(* Logix 5000 project; controller MES_CORE vendor 1 type 14 code 164 rev 32.11; software revision 32.00 *)

TASK MainTask (continuous, watchdog 500 ms) : MES_CORE

MODULES
   Local : vendor 1 type 14 code 164 (ICP 0, rev 32.11)
END_MODULES

VAR_GLOBAL   (* controller tags *)
   ACTIVE_BIT : BOOL;   // FROM LINE
   ANDON : BOOL;   // FROM LINE
   E_STOP : BOOL;   // FROM LINE
   FAULT : BOOL;   // FROM LINE ACTIVE
   JAM_PE : BOOL;   // FROM LINE
   LNXX_ACTIVE_SHIFT : DINT;
   LNXX_SCHEDULE_RUNNING_ONS : BOOL[32];
   LNXX_SCHEDULED_RUN : BOOL;
   LNXX_ShiftChange : BOOL[32];
   LNXX_TO_DC01_DOWNTIME_CODE : DINT[10] := ([0] := 1036); {produced}   // DOWNTIME PRODUCE TAG
        [0]   // LN99
        [1]   // WORK CENTER MAIN LINE A
        [2]   // WORK CENTER MAIN LINE B
        [3]   // WORK CENTER MAIN LINE C
        [4]   // WORK CENTER MAIN LINE D
        [5]   // WORK CENTER MAIN LINE E
        [6]   // WORK CENTER SUB LINE C
        [7]   // WORK CENTER SUB LINE E
   LNXX_TO_DC01_MAIN_MESSAGE : DINT[20] := ([4] := 4480, [16] := 3); {produced}   // KPI PRODUCE TAGS
        [4]   // ACTUAL UNIT COUNT
        [9].0   // LINE RUNNING
        [9].1   // LINE ON BREAK
   LNXX_TO_DC1_MAIN_MESSAGE_A : DINT[10]; {produced}   // WORKCENTER A PRODUCE TAG
        [1]   // LN99NAM01
        [2]   // LN99SAM01
        [3]   // LN99NAM02
        [4]   // LN99SAM02
        [5]   // LN99NAM03
        [6]   // LN99SAM03
        [7]   // LN99NAM04
        [8]   // LN99SAM04
   RUNNING : BOOL;   // FROM LINE
   UNITS_CRATED : DINT;   // FROM LINE
   UNITS_REPAIR : DINT;   // FROM LINE
   WORKSTATION_NUMBER : DINT;   // FROM LINE
END_VAR

PROGRAM MES_CORE   (* main routine MES_MAIN *)
// Cental Team Quality Assurance Environment

ROUTINE _001_IGNITION_DATA_KPI_METRICS   (* ladder *)
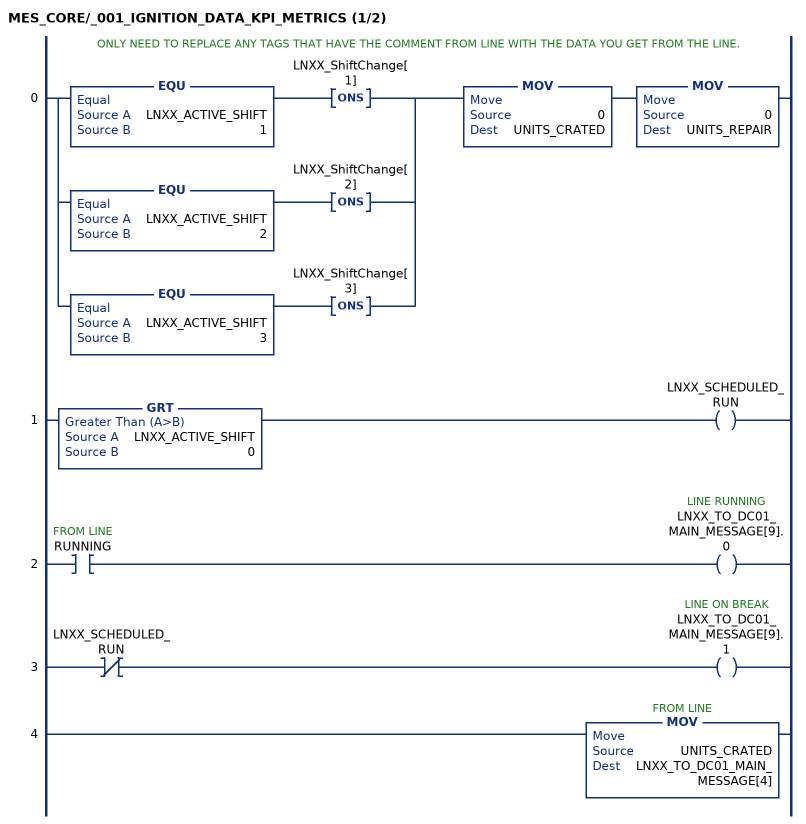
   // ONLY NEED TO REPLACE ANY TAGS THAT HAVE THE COMMENT FROM LINE WITH THE DATA YOU GET FROM THE LINE.
   0: [EQU(LNXX_ACTIVE_SHIFT,1) ONS(LNXX_ShiftChange[1]) ,EQU(LNXX_ACTIVE_SHIFT,2) ONS(LNXX_ShiftChange[2]) ,EQU(LNXX_ACTIVE_SHIFT,3) ONS(LNXX_ShiftChange[3]) ]MOV(0,UNITS_CRATED)MOV(0,UNITS_REPAIR);
   1: GRT(LNXX_ACTIVE_SHIFT,0)OTE(LNXX_SCHEDULED_RUN);
   2: XIC(RUNNING)OTE(LNXX_TO_DC01_MAIN_MESSAGE[9].0);
   3: XIO(LNXX_SCHEDULED_RUN)OTE(LNXX_TO_DC01_MAIN_MESSAGE[9].1);
   4: MOV(UNITS_CRATED,LNXX_TO_DC01_MAIN_MESSAGE[4]);
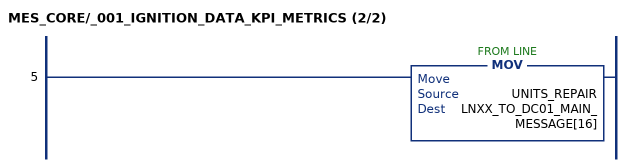
   5: MOV(UNITS_REPAIR,LNXX_TO_DC01_MAIN_MESSAGE[16]);
END_ROUTINE

ROUTINE _002_IGNITION_DATA_OVERALL_MACHINE   (* ladder *)
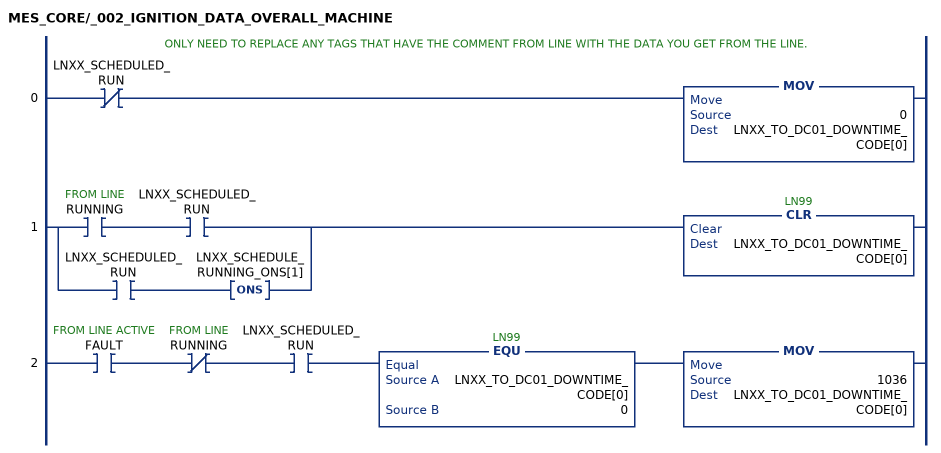
   // ONLY NEED TO REPLACE ANY TAGS THAT HAVE THE COMMENT FROM LINE WITH THE DATA YOU GET FROM THE LINE.
   0: XIO(LNXX_SCHEDULED_RUN)MOV(0,LNXX_TO_DC01_DOWNTIME_CODE[0]);
   1: [XIC(RUNNING) XIC(LNXX_SCHEDULED_RUN) ,XIC(LNXX_SCHEDULED_RUN) ONS(LNXX_SCHEDULE_RUNNING_ONS[1]) ]CLR(LNXX_TO_DC01_DOWNTIME_CODE[0]);
   2: XIC(FAULT)XIO(RUNNING)XIC(LNXX_SCHEDULED_RUN)EQU(LNXX_TO_DC01_DOWNTIME_CODE[0],0)MOV(1036,LNXX_TO_DC01_DOWNTIME_CODE[0]);
END_ROUTINE

ROUTINE _003_IGNITION_DATA_WORKCENTER   (* ladder *)
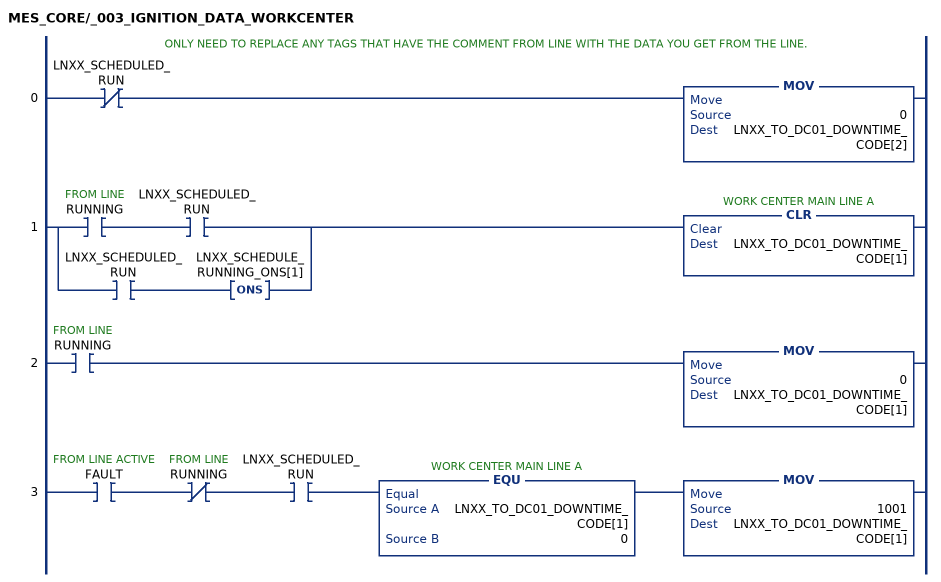
   // ONLY NEED TO REPLACE ANY TAGS THAT HAVE THE COMMENT FROM LINE WITH THE DATA YOU GET FROM THE LINE.
   0: XIO(LNXX_SCHEDULED_RUN)MOV(0,LNXX_TO_DC01_DOWNTIME_CODE[2]);
   1: [XIC(RUNNING) XIC(LNXX_SCHEDULED_RUN) ,XIC(LNXX_SCHEDULED_RUN) ONS(LNXX_SCHEDULE_RUNNING_ONS[1]) ]CLR(LNXX_TO_DC01_DOWNTIME_CODE[1]);
   2: XIC(RUNNING)MOV(0,LNXX_TO_DC01_DOWNTIME_CODE[1]);
   3: XIC(FAULT)XIO(RUNNING)XIC(LNXX_SCHEDULED_RUN)EQU(LNXX_TO_DC01_DOWNTIME_CODE[1],0)MOV(1001,LNXX_TO_DC01_DOWNTIME_CODE[1]);
END_ROUTINE

ROUTINE _004_IGNITION_DATA_WORKSTATION_MAINLINE   (* ladder *)
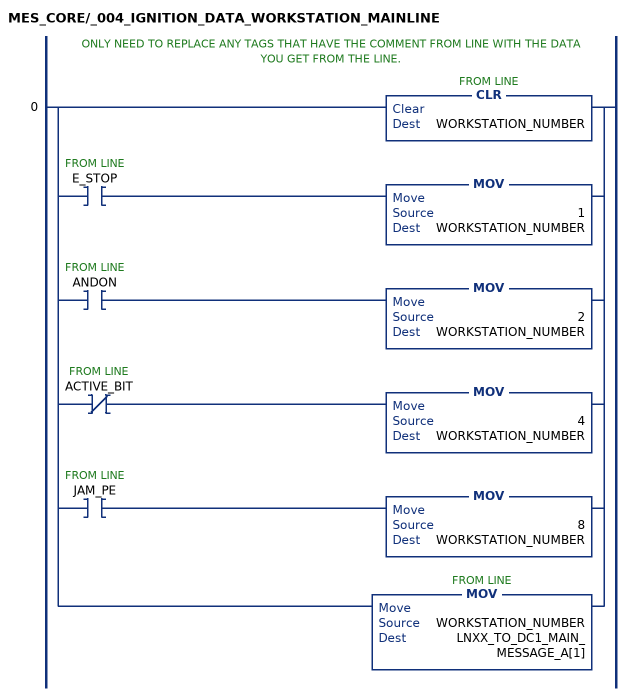
   // ONLY NEED TO REPLACE ANY TAGS THAT HAVE THE COMMENT FROM LINE WITH THE DATA YOU GET FROM THE LINE.
   0: [CLR(WORKSTATION_NUMBER) ,XIC(E_STOP) MOV(1,WORKSTATION_NUMBER) ,XIC(ANDON) MOV(2,WORKSTATION_NUMBER) ,XIO(ACTIVE_BIT) MOV(4,WORKSTATION_NUMBER) ,XIC(JAM_PE) MOV(8,WORKSTATION_NUMBER) ,MOV(WORKSTATION_NUMBER,LNXX_TO_DC1_MAIN_MESSAGE_A[1]) ];
END_ROUTINE

ROUTINE MES_MAIN   (* ladder *)
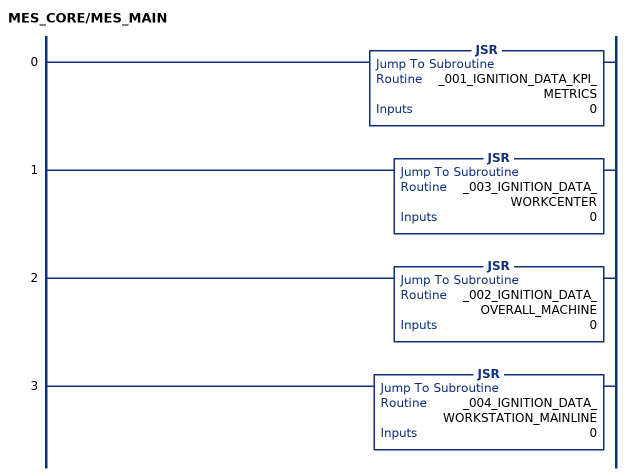
   0: JSR(_001_IGNITION_DATA_KPI_METRICS,0);
   1: JSR(_003_IGNITION_DATA_WORKCENTER,0);
   2: JSR(_002_IGNITION_DATA_OVERALL_MACHINE,0);
   3: JSR(_004_IGNITION_DATA_WORKSTATION_MAINLINE,0);
END_ROUTINE
END_PROGRAM
